TYPE stJoint6 :
STRUCT
	joint1 : LREAL;
	joint2 : LREAL;
	joint3 : LREAL;
	joint4 : LREAL;
	joint5 : LREAL;
	joint6 : LREAL;
END_STRUCT
END_TYPE

(* stored: Version 1.1.0.1, ProductVersion 3.1.4026.18
   DUT stJoint6: Id {b1b2c3d4-1111-1111-1111-111111111111} *)
